// TIA Portal V20 export
TYPE "LER_TypeOffset"
// stored: Access Published
   STRUCT
      SetValue : LReal;
      ProcessValue : LReal;
      UpBtn : Bool;
      DownBtn : Bool;
   END_STRUCT;
END_TYPE
